FUNCTION_BLOCK FB_SubTank_C
VAR_INPUT	
	sublevel					:BOOL;
	protectLevel				:BOOL;	
	filterTime_ON				:TIME;	//接通滤波时间
	filterTime_OFF				:TIME;	//接断开滤波间
	inkFillTimeOutSet			:TIME;   //供墨超时时间设定 s	
END_VAR
VAR_OUTPUT	
	PumpWorking 				:BOOL;	//输出
	state								:INT;
	error_code					:INT;
	Error						:BOOL;
END_VAR
VAR	
	step						:INT;
	ON_filterTon			:TON;						//滤波
	OFF_filterTon			:TON;
	ON_filterTon_P			:TON;						//保护气瓶滤波
	OFF_filterTon_P			:TON;
	filterLevel			    :BOOL;
	filterLevel_P			:BOOL;
	inkFillTimeOutTon		:TON;	
END_VAR
VAR_IN_OUT
	setoff					:BOOL;
END_VAR

ACT_filter_level();

CASE step OF
0://ready
	state:=SubTankStateEnum.ready;
	(************Pumping*****************)
	IF NOT filterLevel AND NOT filterLevel_P  THEN 		
		PumpWorking :=TRUE;
	END_IF	
	IF 	 filterLevel OR  filterLevel_P  THEN
		PumpWorking :=FALSE;
	END_IF
	
	(************inkFillTimeOut*****************)
	inkFillTimeOutTon(IN:=PumpWorking   , PT:=inkFillTimeOutSet , Q=> , ET=> );
		IF inkFillTimeOutTon.Q THEN 
			error_code:=SubTankErrorEnum.pump_timeout;
			step:=100;	
		END_IF	
	
90://setoff
	error:=FALSE;	
	error_code:=ISSErrorEnum.no_error;
		
	inkFillTimeOutTon(IN:=FALSE);
	PumpWorking  :=FALSE;		
	step:=0;		
	
100://error
	state:=SubTankStateEnum.error;
	inkFillTimeOutTon(IN:=FALSE);
	PumpWorking  :=FALSE;	
	error:=TRUE;
END_CASE

IF setoff OR GVL.Reset THEN 
	setoff:=FALSE;
	step:=90;
END_IF
(*****************************************************)
	IF GVL.Emstop_Button  THEN 
		error_code:=ISSErrorEnum.emergency_error;
		step:=100;
	ELSIF filterLevel_P THEN 
		error_code:=ISSErrorEnum.back_to_air_tank;
		step:=100;
	END_IF

ACTION ACT_filter_level:
(************LEVEL*****************)
ON_filterTon(IN:=sublevel , PT:=filterTime_ON , Q=> , ET=> );
OFF_filterTon(IN:=NOT sublevel , PT:=filterTime_OFF , Q=> , ET=> );

IF ON_filterTon .Q  THEN 
	filterLevel:=TRUE;
ELSIF OFF_filterTon .Q THEN 
	filterLevel:=FALSE;
END_IF

(*************LEVEL_P****************)
ON_filterTon_P(IN:=protectLevel , PT:=filterTime_ON , Q=> , ET=> );
OFF_filterTon_P(IN:=NOT protectLevel , PT:=filterTime_OFF , Q=> , ET=> );

IF ON_filterTon_P .Q  THEN 
	filterLevel_P:=TRUE;
ELSIF OFF_filterTon_P .Q THEN 
	filterLevel_P:=FALSE;
END_IF
END_ACTION

END_FUNCTION_BLOCK

(* stored: Version 1.1.0.1, ProductVersion 3.1.4024.11
   POU FB_SubTank_C: Id {1561efcd-af97-4b95-ba98-4d60b540e3ed}, SpecialFunc None
   Action ACT_filter_level: Id {a97605e3-77fc-4768-99bb-9983eb69e9c1} *)
